{attribute 'GeneratedUsingTerminal: EL3632-0000-0022'}
{attribute addProperty BoxType "EL3632-0000-0022"}
{attribute addProperty Id "StartTimeNextLatchAT %I*ULINT8"}
{attribute addProperty CRC "2600321653"}
{attribute addProperty Size "8"}
TYPE NextSync1Time_9AFDC275 EXTENDS InputBase_8311D824 :
STRUCT
	{attribute addProperty Name "StartTimeNextLatch"}
	StartTimeNextLatch AT %I* : ULINT;
END_STRUCT
END_TYPE

(* stored: Version 1.2.0.0, ProductVersion 3.1.4024.9
   DUT NextSync1Time_9AFDC275: Id {2f5e4d94-5096-4c9b-995e-c98172112992} *)
